FUNCTION_BLOCK App1_ReactorPressureandReactorTemp (* Composite Function Block Type *)
  (* Standard: 61499-2 *)
  (* Version 0.0, 2018-11-06, 4DIAC-IDE, 4DIAC-Consortium *)
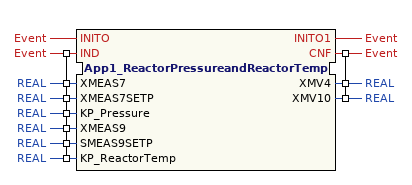
  EVENT_INPUT
    INITO; (* Initialization Request *)
    IND WITH XMEAS7, XMEAS7SETP, KP_Pressure, XMEAS9, SMEAS9SETP, KP_ReactorTemp; (* Normal Execution Request *)
  END_EVENT
  EVENT_OUTPUT
    INITO1; (* Initialization Confirm *)
    CNF WITH XMV4, XMV10; (* Execution Confirmation *)
  END_EVENT
  VAR_INPUT
    XMEAS7 : REAL;
    XMEAS7SETP : REAL;
    KP_Pressure : REAL;
    XMEAS9 : REAL;
    SMEAS9SETP : REAL;
    KP_ReactorTemp : REAL;
  END_VAR
  VAR_OUTPUT
    XMV4 : REAL;
    XMV10 : REAL;
  END_VAR
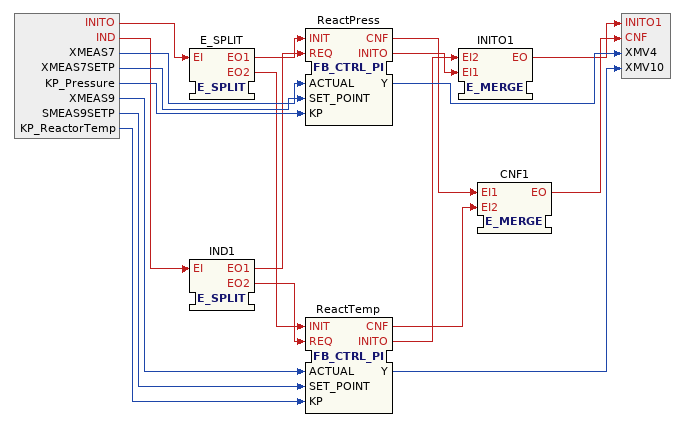
  FBS
    ReactPress : FB_CTRL_PI;
    CNF1 : E_MERGE;
    IND1 : E_SPLIT;
    E_SPLIT : E_SPLIT;
    ReactTemp : FB_CTRL_PI;
    INITO1 : E_MERGE;
  END_FBS
  EVENT_CONNECTIONS
    CNF1.EO TO CNF;
    IND TO IND1.EI;
    INITO TO E_SPLIT.EI;
    E_SPLIT.EO1 TO ReactPress.INIT;
    E_SPLIT.EO2 TO ReactTemp.INIT;
    ReactPress.CNF TO CNF1.EI1;
    ReactTemp.CNF TO CNF1.EI2;
    IND1.EO1 TO ReactPress.REQ;
    IND1.EO2 TO ReactTemp.REQ;
    ReactTemp.INITO TO INITO1.EI2;
    ReactPress.INITO TO INITO1.EI1;
    INITO1.EO TO INITO1;
  END_CONNECTIONS
  DATA_CONNECTIONS
    XMEAS7 TO ReactPress.ACTUAL;
    XMEAS7SETP TO ReactPress.SET_POINT;
    KP_Pressure TO ReactPress.KP;
    ReactPress.Y TO XMV4;
    ReactTemp.Y TO XMV10;
    XMEAS9 TO ReactTemp.ACTUAL;
    SMEAS9SETP TO ReactTemp.SET_POINT;
    KP_ReactorTemp TO ReactTemp.KP;
  END_CONNECTIONS
END_FUNCTION_BLOCK
